// TIA Portal V20 export
FUNCTION_BLOCK "za_TracecodeGeneration_backUp"   // FB35, LAD
TITLE = Tracecode Generation Logic
VERSION : 1.0
// <@VER 1.000>
// Tracecode Generation Logic for J3 Cell Manufacturing specs.
// 26 Char Tracecode
// To be used ONLY in Battery Cell Manufacturing
// stored: MemoryReserve 100, SetENOAutomatically false
   VAR_INPUT
      ComponentType : String;
      MfgSiteId : String;
      Shift : String;
      LineIdentifier : String;
      GMPartNumber : String;
      SignalForTC_Creation : Bool;
      SignalForSN_Increment : Bool;
      SignalForSN_Reset : Bool;
      SignalForTCBuffer_Clear : Bool;
      AlwaysON : Bool;
      ProgramID : String;
      System_Clock_1s_Pulse : Bool;
   END_VAR
   VAR_OUTPUT
      TracebilityCode : String;
      TracebilityCode_Ready : Bool;
   END_VAR
   VAR
      TCtimer : TON_TIME;
   END_VAR
   VAR_TEMP
      RD_Sys_T_RetVal : Int;
      RD_Sys_T_Out : DTL;
      YearinDint : DInt;
      YearinString : String;
      "BulidYear_Decade&Year" : String;
      LGF_CalDay_RetVal : DInt;
      LGF_CalDay_Error : Bool;
      LGF_CalDay_Status : Word;
      DayOfYearinString : String;
      DailySequenceNumber : DInt;
      PulseSN_Increment : Bool;
      PulseSN_Reset : Bool;
      IntermidateString1 : String;
      IntermidateString2 : String;
      IntermidateString3 : String;
      IntermidateString4 : String;
      IntermidateString5 : String;
      InermidateString6 : String;
      DailySequenceNumber_String : String;
      InermidateString7 : String;
      TracebilityCodelocal : String;
      PulseSignalForTC_Creation : Bool;
      TCdone : Bool;
      Pusle1s : Bool;
      TimerCV : Int;
   END_VAR
   VAR_TEMP   // added for the SCL form of the ladder/FBD networks
      _w1 : Bool;
      _w2 : Bool;
      _w3 : Bool;
      _w4 : Bool;
      _w5 : Bool;
   END_VAR
BEGIN

REGION Network 1: Read local time and date
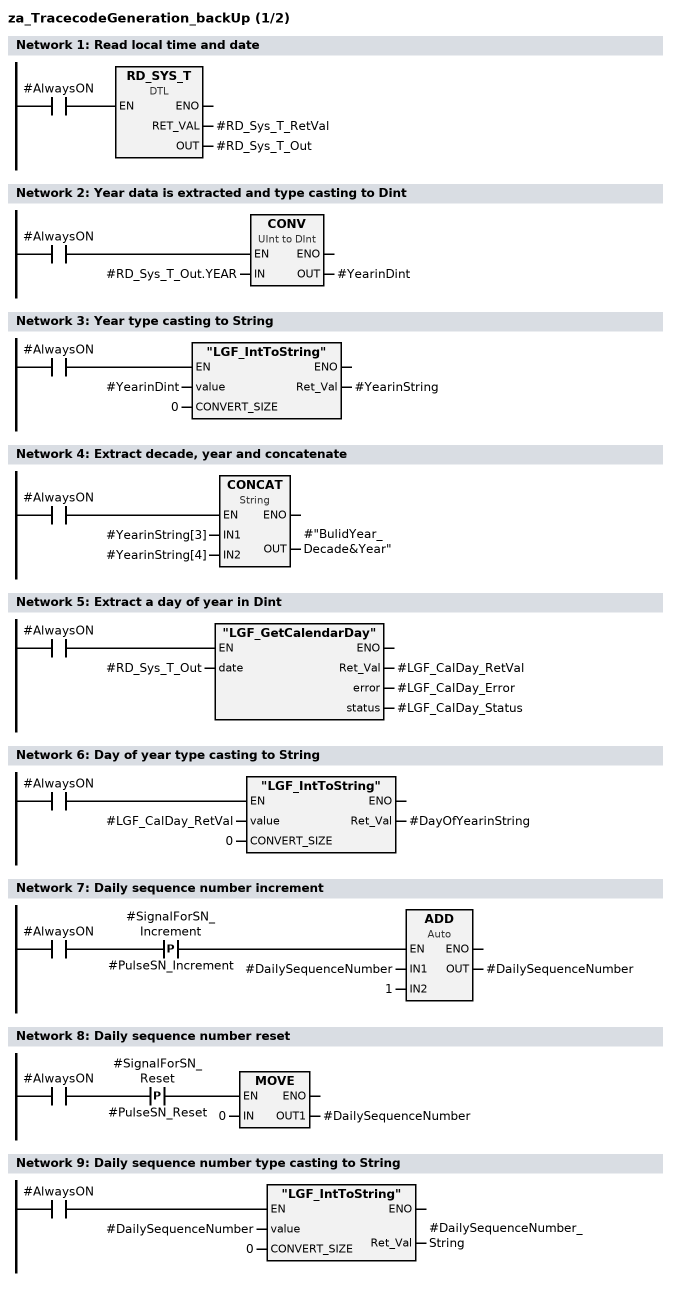
   RUNG wire#powerrail
      Contact( #AlwaysON )
      { S7_Templates := "date_type := DTL" } RD_SYS_T(RET_VAL => #RD_Sys_T_RetVal, OUT => #RD_Sys_T_Out)
   END_RUNG
   // the same network as SCL:
   IF #AlwaysON THEN #RD_Sys_T_RetVal := RD_SYS_T(OUT => #RD_Sys_T_Out); END_IF;
END_REGION

REGION Network 2: Year data is extracted and type casting to Dint
   RUNG wire#powerrail
      Contact( #AlwaysON )
      { S7_Templates := "[SrcType := UInt, DestType := DInt]" } Convert(in := #RD_Sys_T_Out.YEAR, out => #YearinDint)
   END_RUNG
   // the same network as SCL:
   IF #AlwaysON THEN #YearinDint := UINT_TO_DINT(#RD_Sys_T_Out.YEAR); END_IF;
END_REGION

REGION Network 3: Year type casting to String
   RUNG wire#powerrail
      Contact( #AlwaysON )
      "LGF_IntToString"(value := #YearinDint, CONVERT_SIZE := 0, Ret_Val => #YearinString)
   END_RUNG
   // the same network as SCL:
   IF #AlwaysON THEN #YearinString := "LGF_IntToString"(value := #YearinDint, CONVERT_SIZE := 0); END_IF;
END_REGION

REGION Network 4: Extract decade, year and concatenate
   RUNG wire#powerrail
      Contact( #AlwaysON )
      { S7_Templates := "[card := 2, str_type := String]" } CONCAT(IN1 := #YearinString[3], IN2 := #YearinString[4], OUT => #"BulidYear_Decade&Year")
   END_RUNG
   // the same network as SCL:
   IF #AlwaysON THEN
       CONCAT(IN1 := #YearinString[3], IN2 := #YearinString[4], OUT => #"BulidYear_Decade&Year");
   END_IF;
END_REGION

REGION Network 5: Extract a day of year in Dint
   RUNG wire#powerrail
      Contact( #AlwaysON )
      "LGF_GetCalendarDay"("date" := #RD_Sys_T_Out, Ret_Val => #LGF_CalDay_RetVal, error => #LGF_CalDay_Error, status => #LGF_CalDay_Status)
   END_RUNG
   // the same network as SCL:
   IF #AlwaysON THEN
       #LGF_CalDay_RetVal := "LGF_GetCalendarDay"("date" := #RD_Sys_T_Out,
                               error => #LGF_CalDay_Error,
                               status => #LGF_CalDay_Status);
   END_IF;
END_REGION

REGION Network 6: Day of year type casting to String
   RUNG wire#powerrail
      Contact( #AlwaysON )
      "LGF_IntToString"(value := #LGF_CalDay_RetVal, CONVERT_SIZE := 0, Ret_Val => #DayOfYearinString)
   END_RUNG
   // the same network as SCL:
   IF #AlwaysON THEN
       #DayOfYearinString := "LGF_IntToString"(value := #LGF_CalDay_RetVal, CONVERT_SIZE := 0);
   END_IF;
END_REGION

REGION Network 7: Daily sequence number increment
   RUNG wire#powerrail
      Contact( #AlwaysON )
      P_Contact(operand := #SignalForSN_Increment, bit := #PulseSN_Increment)
      Add(in1 := #DailySequenceNumber, in2 := 1, out => #DailySequenceNumber)
   END_RUNG
   // the same network as SCL:
   #_w1 := #AlwaysON AND #SignalForSN_Increment AND NOT #PulseSN_Increment;   // rising edge of #SignalForSN_Increment
   #PulseSN_Increment := #SignalForSN_Increment;
   IF #_w1 THEN #DailySequenceNumber := #DailySequenceNumber + 1; END_IF;
END_REGION

REGION Network 8: Daily sequence number reset
   RUNG wire#powerrail
      Contact( #AlwaysON )
      P_Contact(operand := #SignalForSN_Reset, bit := #PulseSN_Reset)
      Move(in := 0, out1 => #DailySequenceNumber)
   END_RUNG
   // the same network as SCL:
   #_w1 := #AlwaysON AND #SignalForSN_Reset AND NOT #PulseSN_Reset;   // rising edge of #SignalForSN_Reset
   #PulseSN_Reset := #SignalForSN_Reset;
   IF #_w1 THEN #DailySequenceNumber := 0; END_IF;
END_REGION

REGION Network 9: Daily sequence number type casting to String
   RUNG wire#powerrail
      Contact( #AlwaysON )
      "LGF_IntToString"(value := #DailySequenceNumber, CONVERT_SIZE := 0, Ret_Val => #DailySequenceNumber_String)
   END_RUNG
   // the same network as SCL:
   IF #AlwaysON THEN
       #DailySequenceNumber_String := "LGF_IntToString"(value := #DailySequenceNumber, CONVERT_SIZE := 0);
   END_IF;
END_REGION

REGION Network 10: Concanate all data as String
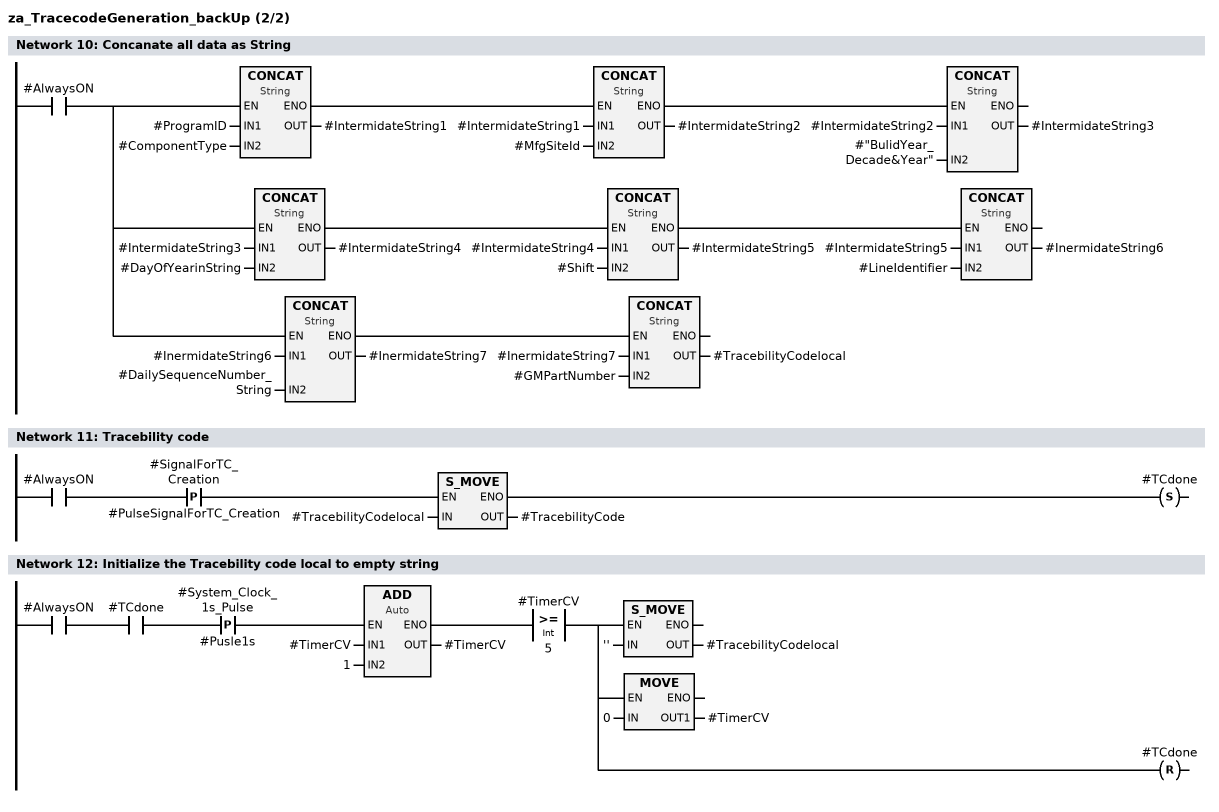
   RUNG wire#powerrail
      Contact( #AlwaysON )
      wire#w1
      { S7_Templates := "[card := 2, str_type := String]" } CONCAT(IN1 := #ProgramID, IN2 := #ComponentType, OUT => #IntermidateString1)
      { S7_Templates := "[card := 2, str_type := String]" } CONCAT(IN1 := #IntermidateString1, IN2 := #MfgSiteId, OUT => #IntermidateString2)
      { S7_Templates := "[card := 2, str_type := String]" } CONCAT(IN1 := #IntermidateString2, IN2 := #"BulidYear_Decade&Year", OUT => #IntermidateString3)
   END_RUNG
   RUNG wire#w1
      { S7_Templates := "[card := 2, str_type := String]" } CONCAT(IN1 := #IntermidateString3, IN2 := #DayOfYearinString, OUT => #IntermidateString4)
      { S7_Templates := "[card := 2, str_type := String]" } CONCAT(IN1 := #IntermidateString4, IN2 := #Shift, OUT => #IntermidateString5)
      { S7_Templates := "[card := 2, str_type := String]" } CONCAT(IN1 := #IntermidateString5, IN2 := #LineIdentifier, OUT => #InermidateString6)
   END_RUNG
   RUNG wire#w1
      { S7_Templates := "[card := 2, str_type := String]" } CONCAT(IN1 := #InermidateString6, IN2 := #DailySequenceNumber_String, OUT => #InermidateString7)
      { S7_Templates := "[card := 2, str_type := String]" } CONCAT(IN1 := #InermidateString7, IN2 := #GMPartNumber, OUT => #TracebilityCodelocal)
   END_RUNG
   // the same network as SCL:
   CONCAT(EN := #AlwaysON, IN1 := #ProgramID, IN2 := #ComponentType, OUT => #IntermidateString1, ENO => #_w1);
   CONCAT(EN := #_w1, IN1 := #IntermidateString1, IN2 := #MfgSiteId, OUT => #IntermidateString2, ENO => #_w2);
   IF #_w2 THEN
       CONCAT(IN1 := #IntermidateString2, IN2 := #"BulidYear_Decade&Year", OUT => #IntermidateString3);
   END_IF;
   CONCAT(EN := #AlwaysON,
          IN1 := #IntermidateString3,
          IN2 := #DayOfYearinString,
          OUT => #IntermidateString4,
          ENO => #_w3);
   CONCAT(EN := #_w3, IN1 := #IntermidateString4, IN2 := #Shift, OUT => #IntermidateString5, ENO => #_w4);
   IF #_w4 THEN
       CONCAT(IN1 := #IntermidateString5, IN2 := #LineIdentifier, OUT => #InermidateString6);
   END_IF;
   CONCAT(EN := #AlwaysON,
          IN1 := #InermidateString6,
          IN2 := #DailySequenceNumber_String,
          OUT => #InermidateString7,
          ENO => #_w5);
   IF #_w5 THEN
       CONCAT(IN1 := #InermidateString7, IN2 := #GMPartNumber, OUT => #TracebilityCodelocal);
   END_IF;
END_REGION

REGION Network 11: Tracebility code
   RUNG wire#powerrail
      Contact( #AlwaysON )
      P_Contact(operand := #SignalForTC_Creation, bit := #PulseSignalForTC_Creation)
      S_Move(in := #TracebilityCodelocal, out => #TracebilityCode)
      S_Coil( #TCdone )
   END_RUNG
   // the same network as SCL:
   #_w1 := #AlwaysON AND #SignalForTC_Creation AND NOT #PulseSignalForTC_Creation;   // rising edge of #SignalForTC_Creation
   #PulseSignalForTC_Creation := #SignalForTC_Creation;
   IF #_w1 THEN
       #TracebilityCode := #TracebilityCodelocal;
       #TCdone := TRUE;
   END_IF;
END_REGION

REGION Network 12: Initialize the Tracebility code local to empty string
   RUNG wire#powerrail
      Contact( #AlwaysON )
      Contact( #TCdone )
      P_Contact(operand := #System_Clock_1s_Pulse, bit := #Pusle1s)
      Add(in1 := #TimerCV, in2 := 1, out => #TimerCV)
      { S7_Templates := "SrcType := Int" } GE_Contact(in1 := #TimerCV, in2 := 5)
      wire#w1
      S_Move(in := '', out => #TracebilityCodelocal)
   END_RUNG
   RUNG wire#w1
      Move(in := 0, out1 => #TimerCV)
   END_RUNG
   RUNG wire#w1
      R_Coil( #TCdone )
   END_RUNG
   // the same network as SCL:
   #_w1 := #AlwaysON AND #TCdone AND #System_Clock_1s_Pulse AND NOT #Pusle1s;   // rising edge of #System_Clock_1s_Pulse
   #Pusle1s := #System_Clock_1s_Pulse;
   IF #_w1 THEN #TimerCV := #TimerCV + 1; END_IF;
   IF #_w1 AND (#TimerCV >= 5) THEN #TracebilityCodelocal := ''; END_IF;
   #_w2 := #_w1 AND (#TimerCV >= 5);
   IF #_w2 THEN
       #TimerCV := 0;
       #TCdone := FALSE;
   END_IF;
END_REGION
END_FUNCTION_BLOCK
